{attribute 'linkalways'} 
{attribute 'no_explicit_call' := 'This FB is a CLASS and must be accessed using methods or properties'}
{attribute 'enable_dynamic_creation'}
FUNCTION_BLOCK FINAL SEL_UDINT EXTENDS Node
VAR
	g : _BOOL(FALSE);
	in1 : _UDINT(0);
	in2 : _UDINT(0);
	out : _UDINT(0);
END_VAR

METHOD PUBLIC Clone : I_Node
VAR
	pNode : POINTER TO SEL_UDINT;
END_VAR
pNode := __NEW(SEL_UDINT);
Clone := pNode^;
END_METHOD

METHOD FB_init : BOOL
VAR_INPUT
	bInitRetains : BOOL; // if TRUE, the retain variables are initialized (warm start / cold start)
	bInCopyCode : BOOL;  // if TRUE, the instance afterwards gets moved into the copy code (online change)
END_VAR
AddInput('g',THIS^.g);
AddInput('in1',THIS^.in1);
AddInput('in2',THIS^.in2);
AddOutput('out', THIS^.out);
END_METHOD

METHOD PROTECTED OnExecute
VAR
END_VAR
IF g.value THEN
	out.value := in2.value;
ELSE
	out.value := in1.value;
END_IF
END_METHOD

END_FUNCTION_BLOCK

(* stored: Version 1.1.0.1, ProductVersion 3.1.4024.15
   POU SEL_UDINT: Id {303c5b4b-2da2-446f-a7a3-0957ceb36074}, SpecialFunc None
   Folder Constructor: Id {9c4a287c-6214-4d1a-9c2a-76cb118807e1}
   Method Clone: Id {ea98c984-e444-4eba-b890-e76d112e918d}
   Method FB_init: Id {8d357645-6d8b-479a-b771-88675d74f343}
   Method OnExecute: Id {33f1ce75-7f9b-4f38-8f50-3161e23fa8b3} *)
